{attribute 'GeneratedUsingTerminal: EK1100-0000-0018'}
{attribute addProperty BoxType "EK1100-0000-0018"}
{attribute addProperty Id "Beckhoff_EL68xxEK1122Beckhoff_EL68xxEK1122_A41DAADD2A_0001_EL6851_0000_0017EL6851_9D5091D6531A_0002_EL6851_0000_0018EL6851_9D5091D6531A_0003_EL6851_0000_0019EL6851_9D5091D6531A_0004_EL6851_0000_0020EL6851_9D5091D6531A_0005_EL6851_0000_0021EL6851_9D5091D6531A_0006_EL6851_0010_0016EL6851_88B184B076A_0007_EL6851_0010_0017EL6851_88B184B076A_0008_EL6851_0010_0018EL6851_88B184B076A_0009_EL6851_0010_0019EL6851_88B184B076A_0010_EL6861_0000_0016EL6861_433C0260274A_0011_EL6861_0000_0017EL6861_433C0260274"}
{attribute addProperty CRC "2680820163"}
{attribute addProperty Size "3509"}
TYPE Beckhoff_EL68xx_9FCA11C3 EXTENDS EK1100_1FC0878B :
STRUCT
	{attribute addProperty Name "Beckhoff_EL68xxEK1122"}
	{attribute addProperty PreviousPort "Beckhoff EL68xx : B"}
	Beckhoff_EL68xxEK1122 : Beckhoff_EL68xxEK1122_A41DAADD;
	{attribute addProperty Name "A_0001_EL6851_0000_0017"}
	{attribute addProperty PreviousPort "Beckhoff EL68xxEK1122 : C"}
	A_0001_EL6851_0000_0017 : EL6851_9D5091D6;
	{attribute addProperty Name "A_0002_EL6851_0000_0018"}
	{attribute addProperty PreviousPort "A_0001(EL6851-0000-0017) : B"}
	A_0002_EL6851_0000_0018 : EL6851_9D5091D6;
	{attribute addProperty Name "A_0003_EL6851_0000_0019"}
	{attribute addProperty PreviousPort "A_0002(EL6851-0000-0018) : B"}
	A_0003_EL6851_0000_0019 : EL6851_9D5091D6;
	{attribute addProperty Name "A_0004_EL6851_0000_0020"}
	{attribute addProperty PreviousPort "A_0003(EL6851-0000-0019) : B"}
	A_0004_EL6851_0000_0020 : EL6851_9D5091D6;
	{attribute addProperty Name "A_0005_EL6851_0000_0021"}
	{attribute addProperty PreviousPort "A_0004(EL6851-0000-0020) : B"}
	A_0005_EL6851_0000_0021 : EL6851_9D5091D6;
	{attribute addProperty Name "A_0006_EL6851_0010_0016"}
	{attribute addProperty PreviousPort "A_0005(EL6851-0000-0021) : B"}
	A_0006_EL6851_0010_0016 : EL6851_88B184B0;
	{attribute addProperty Name "A_0007_EL6851_0010_0017"}
	{attribute addProperty PreviousPort "A_0006(EL6851-0010-0016) : B"}
	A_0007_EL6851_0010_0017 : EL6851_88B184B0;
	{attribute addProperty Name "A_0008_EL6851_0010_0018"}
	{attribute addProperty PreviousPort "A_0007(EL6851-0010-0017) : B"}
	A_0008_EL6851_0010_0018 : EL6851_88B184B0;
	{attribute addProperty Name "A_0009_EL6851_0010_0019"}
	{attribute addProperty PreviousPort "A_0008(EL6851-0010-0018) : B"}
	A_0009_EL6851_0010_0019 : EL6851_88B184B0;
	{attribute addProperty Name "A_0010_EL6861_0000_0016"}
	{attribute addProperty PreviousPort "A_0009(EL6851-0010-0019) : B"}
	A_0010_EL6861_0000_0016 : EL6861_433C0260;
	{attribute addProperty Name "A_0011_EL6861_0000_0017"}
	{attribute addProperty PreviousPort "A_0010(EL6861-0000-0016) : B"}
	A_0011_EL6861_0000_0017 : EL6861_433C0260;
END_STRUCT
END_TYPE

(* stored: Version 1.2.0.0, ProductVersion 3.1.4024.9
   DUT Beckhoff_EL68xx_9FCA11C3: Id {01217c2f-00ef-435b-8d7d-0a8e3095fe25} *)
